(* PLC project , CODESYS GmbH CODESYS V3.5 SP19 *)

TYPE MotorState : (Stopped := 0, Running := 1);
END_TYPE

PROGRAM Main

PROGRAM Main
VAR
    Started : BOOL := TRUE;
END_VAR
END_PROGRAM
END_PROGRAM

CONFIGURATION CfgMain
  RESOURCE ResMain ON PLC
    TASK CyclicTask(INTERVAL := T#100ms, PRIORITY := 1);
  END_RESOURCE
END_CONFIGURATION
